FUNCTION_BLOCK BfbGen
  (* Standard: 61499-2 *)
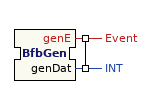
  EVENT_OUTPUT
    genE WITH genDat;
  END_EVENT
  VAR_OUTPUT
    genDat : INT := 1;
  END_VAR
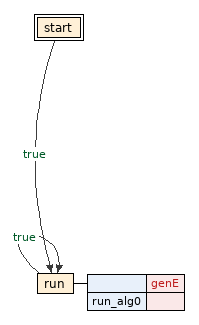
  EC_STATES
    start;
    run : -> genE, run_alg0;
  END_STATES
  EC_TRANSITIONS
    start TO run := true;
    run TO run := true;
  END_TRANSITIONS
  ALGORITHM run_alg0 IN ST:
genDat := genDat + 1;
  END_ALGORITHM
END_FUNCTION_BLOCK
